(* PLC project Senza_nome, Sconosciuto Senza_nome 1 *)
(* stored: creationDateTime 2026-08-24T14:21:44, modificationDateTime 2026-08-24T14:29:48 *)

PROGRAM program0
  VAR
    bt1 AT %IX100.0 : BOOL;
    led AT %QX100.0 : BOOL;
  END_VAR

            
LED := BT1;
          
END_PROGRAM

CONFIGURATION Config0
  RESOURCE Res0 ON PLC
    TASK task0(INTERVAL := T#20ms, PRIORITY := 0);
    PROGRAM instance0 WITH task0 : program0;
  END_RESOURCE
END_CONFIGURATION
